FUNCTION_BLOCK PRESSURE_REGULATOR
VAR_INPUT
	COURANT			: LREAL;
	PRESSION_CONSIGNE : REAL;
	PRESSION_MESURE : REAL;
	MOTOR_POSITION_MAX :FLOAT;
	MOTOR_INITIAL_POSITION: LREAL;
	GEMMA	:STRING;
END_VAR
VAR_OUTPUT
	MOTOR_POSITION 	: DINT;
END_VAR
VAR
	gainScheduled_Kp			: REAL;
	gainScheduled_Ki			: REAL;
	gainScheduled_Kd			: REAL;
	P_ERREUR:REAL;
	GAIN:REAL:=4.0;
	

	eMode						: E_CTRL_MODE;
	stCTRL_PID_PARAMS			: ST_CTRL_PID_PARAMS;

	eErrorId					: E_CTRL_ERRORCODES;
	bError						: BOOL;
	bARWactive					: BOOL;

	(* controller  *)
	fbCTRL_PID					: FB_CTRL_PID;

	fOut: LREAL;
	bHold: BOOL;
END_VAR

IF PUMP_PARAMS.GEN_GRAND_DEBIT=FALSE THEN (*USING STATION 4*)
	IF PRESSION_CONSIGNE>ST4_PID_HighPressure.q THEN
		(*Utilise le régulateur pour les hautes pression*)
		gainScheduled_Kp:=ST4_PID_HighPressure.Kp;
		gainScheduled_Ki:=ST4_PID_HighPressure.Ki;
		gainScheduled_Kd:=ST4_PID_HighPressure.Kd;
	ELSIF PRESSION_CONSIGNE<=ST4_PID_HighPressure.q AND PRESSION_CONSIGNE>ST4_PID_MiddlePressure.q THEN
		(*Calcule les paramètres du régulateur avec une interpolation linéaire entre un PID prévu pour les hautes pressions et un PID pour les moyennes pressions*)
		gainScheduled_Kp:=(ST4_PID_HighPressure.q-PRESSION_CONSIGNE)/(ST4_PID_HighPressure.q-ST4_PID_MiddlePressure.q)*ST4_PID_MiddlePressure.Kp+(PRESSION_CONSIGNE-ST4_PID_MiddlePressure.q)/(ST4_PID_HighPressure.q-ST4_PID_MiddlePressure.q)*ST4_PID_HighPressure.Kp;
		gainScheduled_Ki:=(ST4_PID_HighPressure.q-PRESSION_CONSIGNE)/(ST4_PID_HighPressure.q-ST4_PID_MiddlePressure.q)*ST4_PID_MiddlePressure.Ki+(PRESSION_CONSIGNE-ST4_PID_MiddlePressure.q)/(ST4_PID_HighPressure.q-ST4_PID_MiddlePressure.q)*ST4_PID_HighPressure.Ki;
		gainScheduled_Kd:=(ST4_PID_HighPressure.q-PRESSION_CONSIGNE)/(ST4_PID_HighPressure.q-ST4_PID_MiddlePressure.q)*ST4_PID_MiddlePressure.Kd+(PRESSION_CONSIGNE-ST4_PID_MiddlePressure.q)/(ST4_PID_HighPressure.q-ST4_PID_MiddlePressure.q)*ST4_PID_HighPressure.Kd;
	ELSIF PRESSION_CONSIGNE<=ST4_PID_MiddlePressure.q AND PRESSION_CONSIGNE>ST4_PID_LowPressure.q THEN
		(*Calcule les paramètres du régulateur avec une interpolation linéaire entre un PID prévu pour les moyennes pressions et un PID pour les basses pressions*)
		gainScheduled_Kp:=(ST4_PID_MiddlePressure.q-PRESSION_CONSIGNE)/(ST4_PID_MiddlePressure.q-ST4_PID_LowPressure.q)*ST4_PID_LowPressure.Kp+(PRESSION_CONSIGNE-ST4_PID_LowPressure.q)/(ST4_PID_MiddlePressure.q-ST4_PID_LowPressure.q)*ST4_PID_MiddlePressure.Kp;
		gainScheduled_Ki:=(ST4_PID_MiddlePressure.q-PRESSION_CONSIGNE)/(ST4_PID_MiddlePressure.q-ST4_PID_LowPressure.q)*ST4_PID_LowPressure.Ki+(PRESSION_CONSIGNE-ST4_PID_LowPressure.q)/(ST4_PID_MiddlePressure.q-ST4_PID_LowPressure.q)*ST4_PID_MiddlePressure.Ki;
		gainScheduled_Kd:=(ST4_PID_MiddlePressure.q-PRESSION_CONSIGNE)/(ST4_PID_MiddlePressure.q-ST4_PID_LowPressure.q)*ST4_PID_LowPressure.Kd+(PRESSION_CONSIGNE-ST4_PID_LowPressure.q)/(ST4_PID_MiddlePressure.q-ST4_PID_LowPressure.q)*ST4_PID_MiddlePressure.Kd;
	ELSE (*PRESSION_CONSIGNE<ST4_PID_LowPressure.q*)
		(*Utilise le régulateur pour les basses pressions*)
		gainScheduled_Kp:=ST4_PID_LowPressure.Kp;
		gainScheduled_Ki:=ST4_PID_LowPressure.Ki;
		gainScheduled_Kd:=ST4_PID_LowPressure.Kd;	
	END_IF 
ELSE (*USING STATION 5*)
	(*Utilise le régulateur pour les pressions moyennes*)
	IF PRESSION_CONSIGNE>ST5_PID_MiddlePressure.q THEN
		gainScheduled_Kp:=ST5_PID_MiddlePressure.Kp;
		gainScheduled_Ki:=ST5_PID_MiddlePressure.Ki;
		gainScheduled_Kd:=ST5_PID_MiddlePressure.Kd;	
	ELSIF PRESSION_CONSIGNE<=ST5_PID_MiddlePressure.q AND PRESSION_CONSIGNE>ST5_PID_LowPressure.q THEN
		(*Calcule les paramètres du régulateur avec une interpolation linéaire entre un PID prévu pour les moyennes pressions et un PID pour les basses pressions*)
		gainScheduled_Kp:=(ST5_PID_MiddlePressure.q-PRESSION_CONSIGNE)/(ST5_PID_MiddlePressure.q-ST5_PID_LowPressure.q)*ST5_PID_LowPressure.Kp+(PRESSION_CONSIGNE-ST5_PID_LowPressure.q)/(ST5_PID_MiddlePressure.q-ST5_PID_LowPressure.q)*ST5_PID_MiddlePressure.Kp;
		gainScheduled_Ki:=(ST5_PID_MiddlePressure.q-PRESSION_CONSIGNE)/(ST5_PID_MiddlePressure.q-ST5_PID_LowPressure.q)*ST5_PID_LowPressure.Ki+(PRESSION_CONSIGNE-ST5_PID_LowPressure.q)/(ST5_PID_MiddlePressure.q-ST5_PID_LowPressure.q)*ST5_PID_MiddlePressure.Ki;
		gainScheduled_Kd:=(ST5_PID_MiddlePressure.q-PRESSION_CONSIGNE)/(ST5_PID_MiddlePressure.q-ST5_PID_LowPressure.q)*ST5_PID_LowPressure.Kd+(PRESSION_CONSIGNE-ST5_PID_LowPressure.q)/(ST5_PID_MiddlePressure.q-ST5_PID_LowPressure.q)*ST5_PID_MiddlePressure.Kd;
	ELSE (*PRESSION_CONSIGNE<ST5_PID_LowPressure.q*)
		(*Utilise le régulateur pour les basses pressions*)
		gainScheduled_Kp:=ST5_PID_LowPressure.Kp;
		gainScheduled_Ki:=ST5_PID_LowPressure.Ki;
		gainScheduled_Kd:=ST5_PID_LowPressure.Kd;
	END_IF
END_IF

	(* init parameter struct *)
	stCTRL_PID_PARAMS.tCtrlCycleTime		:= T#10MS;
	stCTRL_PID_PARAMS.tTaskCycleTime		:= T#10MS;
	stCTRL_PID_PARAMS.tTn					:= REAL_TO_TIME(gainScheduled_Ki);			(* integral gain tTn				*)
	stCTRL_PID_PARAMS.tTv					:= REAL_TO_TIME(gainScheduled_Kd);			(* derivative gain tTv				*)
	stCTRL_PID_PARAMS.tTd					:= stCTRL_PID_PARAMS.tTv/5;					(* filter parameter for the real derivative gain part *)
	stCTRL_PID_PARAMS.fKp					:= gainScheduled_Kp;						(* proportional gain Kp				*)
	stCTRL_PID_PARAMS.fOutMaxLimit			:= MOTOR_POSITION_MAX;		  				(* maximum output limit				*)
	stCTRL_PID_PARAMS.fOutMinLimit			:= 0;										(* minimum output limit				*)
	stCTRL_PID_PARAMS.bPInTheFeedbackPath 	:= FALSE;									(* let it to false for a standart PID transfert function *)
    stCTRL_PID_PARAMS.bDInTheFeedbackPath 	:= FALSE;
    stCTRL_PID_PARAMS.bARWOnIPartOnly   	:= TRUE;									(* anti-reset windup *)
	(* set the mode to ACTIVE --> normal operation *)
	eMode							:= eCTRL_MODE_ACTIVE;

	(*Fixe la valeur d'entrée initiale pour le moteur en A1*)
	IF GEMMA = 'A1' THEN
		bHold :=TRUE;
	ELSE
		bHold :=FALSE;
	END_IF

	(*Controller pour la pression*)
	fbCTRL_PID(		fSetpointValue		:= PRESSION_CONSIGNE,
					fActualValue		:= PRESSION_MESURE,
					fManSyncValue		:= MOTOR_INITIAL_POSITION,
					bSync				:= bHold,
					eMode				:= eMode,
					bHold				:= bHold,
					stParams			:= stCTRL_PID_PARAMS,
					fOut				=> fOut,
					bARWactive			=> bARWactive,
					eErrorId			=> eErrorId,
					bError				=> bError
	);
	
MOTOR_POSITION := LREAL_TO_DINT(fOut);



(*	
P_ERREUR:=PRESSION_CONSIGNE - PRESSION_MESURE;

IF COURANT > 10.0 THEN
	MOTOR_POSITION := MOTOR_POSITION + REAL_TO_INT(P_ERREUR*GAIN);(* P_ERREUR*GAIN *)
END_IF;*)

END_FUNCTION_BLOCK

(* stored: Version 1.1.0.1, ProductVersion 3.1.0.26
   POU PRESSURE_REGULATOR: Id {a50045fb-9fcc-4535-9513-631d35e66fe3} *)
